Fanuc KAREL source: kb00124.KL

-- PROVISIONAL review KL for V940-1; original PC SHA256 9b37f5a62deeabac5f6b18d1dbcfe8012983b162bdb3fe79d49b8bff0b630f17
-- Incomplete behavior may be omitted. Consult companion uncertainty JSON. Do not deploy.
PROGRAM KB00124
%NOLOCKGROUP
BEGIN
  -- V9_ZERO_TABLE_METADATA_HINT layout=0002_ascii; no indexed target words; source/name/runtime held
  -- UNRESOLVED_PC offsets 5-14; opcodes 3F,75
  -- UNRESOLVED_PC offsets 19-26; opcodes 9D,23
  -- UNRESOLVED_PC offsets 31-49; opcodes 27,22,2A,22,31
  -- UNRESOLVED_PC offsets 54-58; opcodes 7F
END KB00124
